{attribute 'OPC.UA.DA.StructuredType' := '1'}
FUNCTION_BLOCK FB_Sensor_SICKLevelSwitch_GRF18S EXTENDS FB_BaseDevice IMPLEMENTS I_Device, I_Sensor

VAR
	
	{attribute 'OPC.UA.DA' := '0'} 
	eSensorType: E_SensorType;
	{attribute 'OPC.UA.DA' := '0'} 
	nRawInput AT %I*: BOOL;
	{attribute 'OPC.UA.DA' := '1'} 
	nCurrentValue: REAL;
END_VAR

calculate();

METHOD calculate : BOOL
VAR_INPUT
END_VAR
IF nRawInput THEN
	nCurrentValue := 1;
ELSE
	nCurrentValue := 0;
END_IF
END_METHOD

{warning 'add method implementation '}
METHOD disable : BOOL
bEnable := FALSE;
END_METHOD

{warning 'add method implementation '}
METHOD enable : BOOL
bEnable := TRUE;
END_METHOD

{warning 'add method implementation '}
METHOD FB_init : BOOL
VAR_INPUT
	(* if TRUE, the retain variables are initialized (warm start / cold start)*)
	bInitRetains	: BOOL;
	(* if TRUE, the instance afterwards gets moved into the copy code (online change)*)
	bInCopyCode	: BOOL;
	SensorID	: STRING(80);
	SensorDescr	: STRING(255);
	SensorType	: E_SensorType;
END_VAR
sID := SensorID;
sDescr := SensorDescr;
eSensorType := SensorType;
END_METHOD

{warning 'add method implementation '}
METHOD getType : E_SensorType
getType := eSensorType;
END_METHOD

{warning 'add method implementation '}
METHOD getValue : REAL
getValue := nCurrentValue;
END_METHOD

{warning 'add method implementation '}
METHOD write : BOOL
calculate();
END_METHOD

END_FUNCTION_BLOCK

(* stored: Version 1.1.0.1, ProductVersion 3.1.4024.12
   POU FB_Sensor_SICKLevelSwitch_GRF18S: Id {f45d52d0-7769-4b43-a8f0-30f5a7d78fca}, SpecialFunc None
   Method calculate: Id {76eb7f5f-8eaf-4d43-8455-8a226267a653}
   Method disable: Id {50a73936-121d-4bfe-ac2d-b27e10298248}
   Method enable: Id {b92a0c8a-823c-4a4a-9bc0-6aad587f43ed}
   Method FB_init: Id {c4d13cd2-22f7-4061-9d38-a14bc3138985}
   Method getType: Id {baff93f6-135b-432a-bc7b-20b74e67413b}
   Method getValue: Id {9cf098c1-ea0d-4a0e-8879-4322ce9f5bca}
   Method write: Id {fc9cb89d-fa06-4e94-bf0c-4d28f9b52e59} *)
